(* CoDeSys 2.3 export: COMPOSEINT.EXP *)

(* POU Functions/ComposeInt, ST *)
FUNCTION ComposeInt : INT
VAR_INPUT
	Ones : INT ;
	Tens : INT ;
	Hundreds : INT ;
	Thousands : INT ;
END_VAR
VAR
END_VAR
ComposeInt := (Thousands * 1000) + (Hundreds * 100) + (Tens * 10) + Ones;
END_FUNCTION
